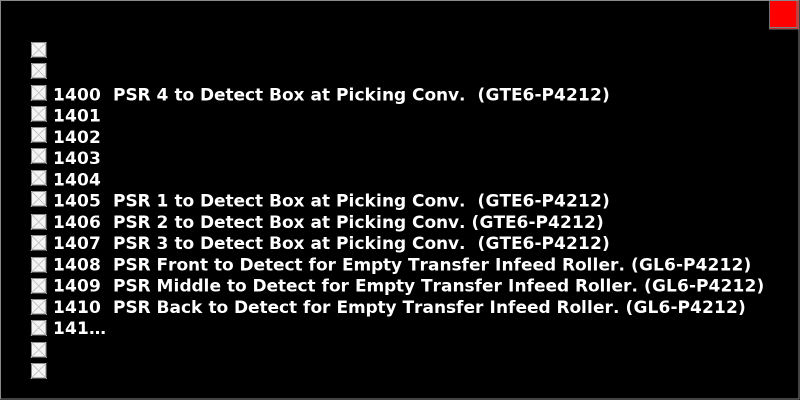
VISUALIZATION P1_DI3  // 800x400, background image 
    ImageSwitcher (31,42 15x15), variable: InputOutput_GVL.xIn1400, behaviour: TOGGLE
    Label (50,16 732x391), "1400 PSR 4 to Detect Box at Picking Conv. (GTE6-P4212) 1401 1402 1403 1404 1405 PSR 1 to Detect Box at Picking Conv. (GTE6-P4212) 1406 PSR 2 to Detect Box at Picking Conv. (GTE6-P4212) 1407 PSR 3 to Detect Box at Picking Conv. (GTE6-P4212) 1408 PSR Front to Detect for Empty Transfer Infeed Roller. (GL6-P4212) 1409 PSR Middle to Detect for Empty Transfer Infeed Roller. (GL6-P4212) 1410 PSR Back to Detect for Empty Transfer Infeed Roller. (GL6-P4212) 1411 1412 1413 1414 Request Release Solenoid Door Robot 1415 Feedback Relay Solenoid Door Robot"
    ImageSwitcher (31,63 15x15), variable: InputOutput_GVL.xIn1401, behaviour: TOGGLE
    ImageSwitcher (31,85 15x15), variable: InputOutput_GVL.xIn1402, behaviour: TOGGLE
    ImageSwitcher (31,106 15x15), variable: InputOutput_GVL.xIn1403, behaviour: TOGGLE
    ImageSwitcher (31,127 15x15), variable: InputOutput_GVL.xIn1404, behaviour: TOGGLE
    ImageSwitcher (31,148 15x15), variable: InputOutput_GVL.xIn1405, behaviour: TOGGLE
    ImageSwitcher (31,170 15x15), variable: InputOutput_GVL.xIn1406, behaviour: TOGGLE
    ImageSwitcher (31,191 15x15), variable: InputOutput_GVL.xIn1407, behaviour: TOGGLE
    ImageSwitcher (31,214 15x15), variable: InputOutput_GVL.xIn1408, behaviour: TOGGLE
    ImageSwitcher (31,235 15x15), variable: InputOutput_GVL.xIn1409, behaviour: TOGGLE
    ImageSwitcher (31,257 15x15), variable: InputOutput_GVL.xIn1410, behaviour: TOGGLE
    ImageSwitcher (31,278 15x15), variable: InputOutput_GVL.xIn1411, behaviour: TOGGLE
    ImageSwitcher (31,299 15x15), variable: InputOutput_GVL.xIn1412, behaviour: TOGGLE
    ImageSwitcher (31,320 15x15), variable: InputOutput_GVL.xIn1413, behaviour: TOGGLE
    ImageSwitcher (31,342 15x15), variable: InputOutput_GVL.xIn1414, behaviour: TOGGLE
    ImageSwitcher (31,363 15x15), variable: InputOutput_GVL.xIn1415, behaviour: TOGGLE
    Button (769,-1 30x30), image: VisuSymbols.Symbols.Wrong
        OnMouseClick: CloseDialog Dialog=P1_DI3, Result=OK, NumpadKeypadSet=True
END_VISUALIZATION

(* stored: Version 1.1.0.1, ProductVersion 3.1.4024.12
   Visu P1_DI3: Id {a2d1076d-978d-4589-9929-d77ebf7113b5} *)
